// Core §8.12 — platform-neutral probe sample. Availability is explicit so an
// unsupported metric never masquerades as a healthy zero.
TYPE ST_SystemHealthInput :
STRUCT
    TaskAvailable       : BOOL;
    TaskCycleUs         : UDINT;
    TaskJitterUs        : UDINT;
    TaskOverrun         : BOOL;
    ControllerAvailable : BOOL;
    CpuLoadPct          : LREAL;
    MemoryAvailableMb   : UDINT;
    IpcAvailable        : BOOL;
    IpcTemperatureC     : LREAL;
    FanHealthy          : BOOL;
    StorageHealthPct    : LREAL;
    FieldbusAvailable   : BOOL;
    FieldbusMasterHealthy : BOOL;
    LostFrameCount      : UDINT;
    SlaveErrorCount     : UDINT;
    DcAvailable         : BOOL;
    DcSynchronized      : BOOL;
    TimeQuality         : ST_TimeQuality;
    // Per-metric availability inside the IPC group (Core §8.12: "where the hardware
    // exposes them"). TRUE by default, so a producer that sets only IpcAvailable
    // keeps its meaning; a target provider clears the one it cannot measure - a
    // fanless IPC, a drive without flash wear data - instead of inventing a value.
    FanAvailable        : BOOL := TRUE;
    StorageAvailable    : BOOL := TRUE;
END_STRUCT
END_TYPE

(* stored: Version 1.1.0.1, ProductVersion 3.1.4024.12
   DUT ST_SystemHealthInput: Id {89f432bb-457e-4500-a84b-1c481fdde476} *)
